{attribute 'linkalways'}
{attribute 'no_explicit_call' := 'do not call this POU directly'}
{attribute 'enable_dynamic_creation'}
FUNCTION_BLOCK JsonPathElement_Property EXTENDS JsonPathElement 
VAR
	name : T_MAXSTRING;
END_VAR

METHOD FB_init : BOOL
VAR_INPUT
	bInitRetains : BOOL; // if TRUE, the retain variables are initialized (warm start / cold start)
	bInCopyCode : BOOL;  // if TRUE, the instance afterwards gets moved into the copy code (online change)
	PreviousElement : I_JsonPathElement;
	NextElement : I_JsonPathElement; 
	Name : T_MAXSTRING;
END_VAR
This^.name := Name;
END_METHOD

PROPERTY PUBLIC PropertyName : T_MAXSTRING
GET
PropertyName := name;
END_GET
END_PROPERTY

METHOD PUBLIC ResolveToSJsonValue : SJsonValue
VAR_INPUT
	jsonParser : REFERENCE TO FB_JsonDomParser;
	jsonDocument : SJsonValue;
END_VAR
VAR
	currentPosition : SJsonValue;
	memberPath : SJsonValue;
END_VAR
IF PreviousElement <> 0 THEN
	currentPosition := PreviousElement.ResolveToSJsonValue(jsonParser,jsonDocument);
ELSE
	currentPosition := jsonDocument;
END_IF

IF currentPosition = 0 THEN
	RETURN;
END_IF

ResolveToSJsonValue := jsonParser.FindMember(currentPosition,name);
END_METHOD

END_FUNCTION_BLOCK

(* stored: Version 1.1.0.1, ProductVersion 3.1.4024.12
   POU JsonPathElement_Property: Id {2f07aa6b-bb05-4d2a-a467-58ebc4bd0cdf}, SpecialFunc None
   Folder Constructor: Id {1bd34833-3f2a-43e6-9e2b-60a4f71cc417}
   Method FB_init: Id {84410c23-ba03-4bf2-a082-e62c128e7c6b}
   Property PropertyName: Id {d027bbab-9864-4dbc-86cb-9f2d180b8163}
   Get Get: Id {1bfe8cff-1019-4b61-8ae7-c975d06daab5}
   Method ResolveToSJsonValue: Id {c28e31bc-d8d4-44b2-94ee-32052359f811} *)
